// TIA Portal V20 export
VAR_GLOBAL   // PLC tag table "Safety tags"
   "MCC001+Phase Sequence Ok" AT %I3.0 : Bool;
   "ZONA1+A1.1.1-SF01" AT %I0.0 : Bool;
   "ZONA1+A1.1.10-SF01" AT %I0.1 : Bool;
   "ZONA1+A1.2.1-SF01" AT %I0.2 : Bool;
   "ZONA1+C1.2.2-SF01" AT %I0.3 : Bool;
   "ZONA1+B0.2.0-SF01" AT %I0.4 : Bool;
   "ZONA1+B1.15.1-SF01" AT %I0.5 : Bool;
   "ZONA1+E1.1.1-SF01" AT %I0.6 : Bool;
   "ZONA2+D1.11.1-SF01" AT %I0.7 : Bool;
   "ZONA2+A1.10.3-SF01" AT %I1.0 : Bool;
   "ZONA2+A1.12.1-SF01" AT %I1.1 : Bool;
   "ZONA2+A1.14.7-SF01" AT %I1.2 : Bool;
   "ZONA2+A1.15.0-SF01" AT %I1.3 : Bool;
   "ZONA2+A2.3.0-SF01" AT %I1.4 : Bool;
   "ZONA2+A2.2.7-SF01" AT %I1.5 : Bool;
   "ZONA2+A2.1.1-SF01" AT %I1.6 : Bool;
   "ZONA2+G1.5.1-SF01" AT %I1.7 : Bool;
   "ZONA1+MCC001-QA1" AT %Q0.0 : Bool;
   "ZONA1+MCC001-QA2" AT %Q0.1 : Bool;
   "ZONA2+MCC001-QA1" AT %Q0.2 : Bool;
   "ZONA2+MCC001-QA2" AT %Q0.3 : Bool;
   Reserved_1 AT %Q0.4 : Bool;
   Reserved_2 AT %Q0.5 : Bool;
   Reserved_3 AT %Q0.6 : Bool;
   Reserved_4 AT %Q0.7 : Bool;
   "ZONA1+Mushiny-QA1" AT %Q1.0 : Bool;
   "ZONA1+Mushiny-QA2" AT %Q1.1 : Bool;
   "Reserved_1(1)" AT %Q1.2 : Bool;
   "Reserved_2(1)" AT %Q1.3 : Bool;
   "Reserved_3(1)" AT %Q1.4 : Bool;
   "Reserved_4(1)" AT %Q1.5 : Bool;
   "Reserved_5(1)" AT %Q1.6 : Bool;
   "ZONA2+G1.7.4-SF01" AT %I2.0 : Bool;
   "MCC001-SF1" AT %I2.1 : Bool;
   "Emergency-Mushiny-1" AT %I2.2 : Bool;
   "Emergency-Mushiny-2" AT %I2.3 : Bool;
   "BPR-FireSafety-1" AT %I2.4 : Bool;
   "BPR-FireSafety-2" AT %I2.5 : Bool;
   Reserve_1 AT %I2.6 : Bool;
   Reserve_2 AT %I2.7 : Bool;
   "Reserved_6(1)" AT %Q1.7 : Bool;
   "Contactor -fb -QA1 -Zone1 -MCC001" AT %I7.6 : Bool;
   "Contactor -fb -QA2 -Zone1 -MCC001" AT %I7.7 : Bool;
   "Contactor -fb -QA1 -Zone2 -MCC001" AT %I8.0 : Bool;
   "Contactor -fb -QA2 -Zone2 -MCC001" AT %I8.1 : Bool;
END_VAR
